{attribute 'qualified_only'}
{attribute 'strict'}
{attribute 'to_string'}
TYPE Modus :
(
	Auto := 0,
	Manual,
	Stop
);
END_TYPE

(* stored: Version 1.1.0.1
   DUT Modus: Id {bd383948-cf02-485c-b3b4-fda68b408657} *)
